PROGRAM MQTT
VAR
// Local Variables for Mqtt Client handling
	fbIotMqttClient : FB_IotMqttClient;
	bSetParameter 	: BOOL := TRUE;
	bConnect 		: BOOL := TRUE;	
	
// Publish message
	initMQTT : BOOL := FALSE;
	sTopicPubToPowerMgmt : STRING(255); //:= CONCAT('Robots/PowerMgmt/Robot_', INT_TO_STRING(.Var_HAWIno.Robot_Number)); 	// ToDo: Bisher ist die Nummer des HAWino fest kodiert
	sTopicPubToPowerMgmt_SOC : STRING(255);// := CONCAT('Robots/PowerMgmt/SoC_Robot_', INT_TO_STRING(.Var_HAWIno.Robot_Number)); 
	sPayloadPub : STRING(2000);	
	fbTimerPub 	: TON := (PT:=T#500MS);									// Intervall für das Senden des Akku-Status
	
//Received message
	bSubscribed    : BOOL;
	sTopicSubToPowerMgmt : STRING(255);// := CONCAT('PowerMgmt/Robots/Robot_', INT_TO_STRING(.Var_HAWIno.Robot_Number));	// ToDo: Bisher ist die Nummer des HAWino fest kodiert
	sTopicRcv      : STRING(255);
	sPayloadRcv    : STRING(255);
	sPayloadRcv_Status    : STRING(255);
	sPayloadRcv_Status_Test: STRING(255);
	fbMessageQueue : FB_IotMqttMessageQueue;
    fbMessage      : FB_IotMqttMessage;
	hrErrorOccurred : HRESULT; 			// Enthlt dern letzten augetretenen Fehler
	
//subscribe
	sTopicSubToGW1_Status : STRING(255);
	sTopicSubToGW1_Auftrag : STRING(255);
	sTopicSubCollision : STRING(255);
	sTopicPubCollision : ARRAY[1..4] OF STRING(255);
	sTopicSubReset : STRING(255);
	
// Variables for JSON
	fbJson			: FB_JsonSaxWriter;
	fbJsonDataType 	: FB_JsonReadWriteDataType;
	sJsonDoc       	: STRING(2000); 
	
// Local Variables for TwinCAT IoT Communication (TF6701) with direct link to EK1200 and TcCom
	//stMqtt_HAWino_In	AT%I*	: ST_PwrMgmt_HAWino_In;		// Attention! Don't link TIME Variables, otherwise we get an error!
	//stMqtt_HAWino_Out	AT%Q*	: ST_PwrMgmt_HAWino_Out;
	
	stMqtt_HAWino_In	 AT%I*: ST_PwrMgmt_HAWino_In;		// Attention! Don't link TIME Variables, otherwise we get an error!
	stMqtt_HAWino_Out	 AT%Q*: ST_PwrMgmt_HAWino_Out;
	
	SOC_Out : STRING(255);
	nBatteryTemperature	AT%I*	: INT;
	
	bComCheckAnswer	AT%Q*	: BOOL;
	
	stMqtt_HAWinoValues	: ST_PwrMgmt_HAWino;
	
	
// Timer to create a time stamp
	fbTimerTimestamp : TON := (PT:=T#71582M47S295MS);
	
// Local Vaiables to evaluate and act to input
	fbComCheckFlag	: RS;
	
	sTopicSubToFleetMgmt: STRING;
	Reset1: BOOL;
	//Input synccheck. robotdata has been read and can be used.
	txtReadInit AT%I* : BOOL := FALSE;
	
	//eigene Topics und Payload
	sTopicPubToGW1 : STRING(255);
	WerkstueckAusgelesen: BOOL;
	sPayloadPub1 : STRING(2000);
	Robotstatus : RobotStatusGW1;
	sTopicSubToGW1: STRING(255);
	nPayloadSize:INT;
	sPayloadPubCollision : STRING(100);
	n: INT;												
	
	FeedbackToGW1 AT%I*: STRING(50);				//Statusmeldungen an Gewerk 1
	RoboNmbToGoBack AT%I* : ARRAY[0..4] OF INT;		//Nummer, der Roboter, die zurück sollen
	resetVar, resetGoBack AT%I*: BOOL;				//Reset Variablen, um Ausgänge zurückzusetzen
	Auftrag AT%Q*: Auftrag;							//Auftrag von Gewerk 1 gesendet
	StatusFromGW1 AT%Q*: STRING(50);				//Statusrückmeldungen von Gewerk 1 gesendet
	goBack AT%Q* : BOOL;							//true, wenn Roboter Platz machen soll
	resetButton AT%Q* : BOOL;						//Reset von Gewerk 1 kommend
END_VAR

//Case machen! preop op

//Unsere Topics und erwartete Struktur:
//Auftrag: {"Art":"Fahrauftrag","AbholStation":1,"AbholTasche":2,"AblageStation":3,"AblageTasche":1}
//Status: {"Status":"WerkstueckAusgelesen"}
//Kollision: {"todo":"goBack"}

IF txtReadInit THEN
	IF NOT initMQTT THEN
		sTopicPubToPowerMgmt  := CONCAT('Robots/PowerMgmt/Robot_', INT_TO_STRING(.Var_HAWIno.Robot_Number)); 	
		sTopicPubToPowerMgmt_SOC  := CONCAT('Robots/PowerMgmt/SoC_Robot_', INT_TO_STRING(.Var_HAWIno.Robot_Number)); 
		sTopicSubToPowerMgmt  := CONCAT('PowerMgmt/Robots/Robot_', INT_TO_STRING(.Var_HAWIno.Robot_Number));
		sTopicSubToGW1  := CONCAT('VPJ/Robot_', INT_TO_STRING(.Var_HAWIno.Robot_Number));
		sTopicSubToGW1_Status  := CONCAT(sTopicSubToGW1, '/Status');
		sTopicSubToGW1_Auftrag  := CONCAT(sTopicSubToGW1, '/Auftrag');
		sTopicPubToGW1 := CONCAT('VPJ/Robot_', INT_TO_STRING(.Var_HAWIno.Robot_Number));
		sTopicSubCollision := CONCAT('VPJ/Robot_', INT_TO_STRING(.Var_HAWIno.Robot_Number));
		sTopicSubCollision := CONCAT(sTopicSubCollision, '/Collision');
		sTopicSubReset  := CONCAT('VPJ/Robot_', INT_TO_STRING(.Var_HAWIno.Robot_Number));
		sTopicSubReset  := CONCAT(sTopicSubToGW1, '/Reset');
		FOR n := 1 TO 4 BY 1 DO
			IF n <> .Var_HAWIno.Robot_Number THEN
				sTopicPubCollision[n] := CONCAT('VPJ/Robot_', INT_TO_STRING(n));
				sTopicPubCollision[n] := CONCAT(sTopicPubCollision[n], '/Collision');
			END_IF
		END_FOR
		initMQTT:= TRUE;
	END_IF
	
	stMqtt_HAWinoValues.Output.nRobotNumber := .Var_HAWIno.Robot_Number;			// Anpassen für jeden HAWino
	
	fbTimerTimestamp(In:= NOT fbTimerTimestamp.Q, ET=>stMqtt_HAWinoValues.Output.tTimestamp);
	
	stMqtt_HAWinoValues.Output.fSoC := stMqtt_HAWino_In.fSoC;
	
	stMqtt_HAWinoValues.Output.fActualBatteryCurrent := stMqtt_HAWino_In.fActualBatteryCurrent;
	stMqtt_HAWinoValues.Output.fActualBatteryVoltage := stMqtt_HAWino_In.fActualBatteryVoltage;

	
	// Skalierung der Temperaturwerte des Akkus
	stMqtt_HAWinoValues.Output.fBatteryTemperature := FKT_Scale(Rohwert := nBatteryTemperature, 
																	X1 := -500,
																	X2 := 1500, 
																	Y1 := -50,
																	Y2 := 150);
																	
	// Ausgabe der erwarteten Laufzeit des Roboters
	stMqtt_HAWinoValues.Output.nEstimatedRunningTime	:= LIMIT(0,stMqtt_HAWino_In.nEstimatedRunningTime,172800);		// Max. 48 Stunden sollen dargestellt werden
	stMqtt_HAWinoValues.Output.nEstimatedChargingTime	:= LIMIT(0,stMqtt_HAWino_In.nEstimatedChargingTime,172800);		// Max. 48 Stunden sollen dargestellt werden
	
	
	// Antworten auf den Kommunikationstest und des Ladetests
	stMqtt_HAWinoValues.Output.bCheckCurrentDetected := stMqtt_HAWino_In.bCheckCurrentDetected;
	stMqtt_HAWinoValues.Output.bComCheckAnswer := stMqtt_HAWino_In.bComCheckAnswer;
	
	//
	// Setting the parameters for establishing the connection to the Mqtt Broker and initializing the connection.
	//
	IF bSetParameter THEN
		fbIotMqttClient.sHostName := '192.168.0.11';	// IP-Adresse des Servers
		fbIotMqttClient.nHostPort := 1883;
		//fbIotMqttClient.sClientId := ClientId;
		fbIotMqttClient.sClientId := CONCAT('Robot_', INT_TO_STRING(.Var_HAWIno.Robot_Number));
		fbIotMqttClient.sTopicPrefix := '';
		//fbIotMqttClient.nKeepAlive:= 60; 
		fbIotMqttClient.sUserName:= 'VPJ';
		fbIotMqttClient.sUserPassword:= 'R462';
		//fbIotMqttClient.stWill:= ; 
		//fbIotMqttClient.stTLS:= ;
		fbIotMqttClient.ipMessageQueue := fbMessageQueue;
	
		bSetParameter := FALSE;
	END_IF
	
	
	//
	// This method -> MUST BE CALLED CYCLICALLY <- to ensure background communication with the MQTT broker.
	//
	fbIotMqttClient.Execute(bConnect);
	
	IF fbIotMqttClient.bError THEN
		// ToDo: add error logging here
		hrErrorOccurred := fbIotMqttClient.hrErrorCode;
	END_IF
	
		
	IF fbIotMqttClient.bConnected THEN		// Kontrolle, ob der Broker verbunden ist
		IF NOT bSubscribed THEN
			//
			// Abbonieren der Toopics, welche vom PowerMgmt kommen
			//
			bSubscribed := fbIotMqttClient.Subscribe(sTopic:=sTopicSubToPowerMgmt, eQoS:=TcIotMqttQos.AtMostOnceDelivery);
			IF fbIotMqttClient.bError THEN
				// ToDo: add my error logging here
				hrErrorOccurred := fbIotMqttClient.hrErrorCode;
			END_IF
			
			//
			// Abbonieren der Toopics, welche vom Gewerk 1 kommen
			//
			//Abbonieren von Topics: VPJ/Roboter
			bSubscribed := fbIotMqttClient.Subscribe(sTopic:=sTopicSubToGW1_Status, eQoS:=TcIotMqttQos.AtMostOnceDelivery);
			bSubscribed := fbIotMqttClient.Subscribe(sTopic:=sTopicSubToGW1_Auftrag, eQoS:=TcIotMqttQos.AtMostOnceDelivery);
			bSubscribed := fbIotMqttClient.Subscribe(sTopic:=sTopicSubCollision, eQoS:=TcIotMqttQos.AtMostOnceDelivery);
			bSubscribed := fbIotMqttClient.Subscribe(sTopic:=sTopicSubReset, eQoS:=TcIotMqttQos.AtMostOnceDelivery);
			
			
			//bSubscribed := fbIotMqttClient.Subscribe(sTopic:=sTopicSubToFleetMgmt, eQoS:=TcIotMqttQos.AtMostOnceDelivery);
			//IF fbIotMqttClient.bError THEN
				// ToDo: add my error logging here
			//	hrErrorOccurred := fbIotMqttClient.hrErrorCode;
			//END_IF
			
		END_IF
	END_IF	
	
	
	
	// Senden der MQTT- Nachrichten
	
	
	IF fbIotMqttClient.bConnected THEN			// Kontrolle, ob Broker verbunden ist
		fbTimerPub(IN:=TRUE);
		
		//
		// publish new paylod every 500 MS
		//
		IF fbTimerPub.Q THEN					// Abwarten des oben eingestellten Intervalls
			fbTimerPub(IN:=FALSE);
			
			//
			// Nachricht an PowerMgmt
			//
			fbJson.ResetDocument();
			fbJsonDataType.AddJsonValueFromSymbol(fbJson, 'ST_PwrMgmt_HAWino_In', SIZEOF(stMqtt_HAWinoValues.Output), ADR(stMqtt_HAWinoValues.Output));
			//sJsonDoc := fbJson.GetDocument();
			fbJson.CopyDocument(sJsonDoc, SIZEOF(sJsonDoc));
			
			sPayloadPub := sJsonDoc;	
			fbIotMqttClient.Publish(sTopic:= sTopicPubToPowerMgmt, 
										pPayload:= ADR(sPayloadPub), 
										nPayloadSize:= LEN2(ADR(sPayloadPub))+1, 										
										eQoS:= TcIotMqttQos.AtMostOnceDelivery, 
										bRetain:= FALSE, 
										bQueue:= FALSE);
									
									
			
			SOC_Out	:= CONCAT( '{"SoC" : ',LREAL_TO_STRING(stMqtt_HAWinoValues.Output.fSoC));
			SOC_Out	:= CONCAT( SOC_Out,'}');
			
			
			
			
			//SOC_Out := 	LREAL_TO_STRING(stMqtt_HAWinoValues.Output.fSoC);
			
						
			fbIotMqttClient.Publish(sTopic:= sTopicPubToPowerMgmt_SOC, 
										pPayload:=ADR(SOC_Out), 
										nPayloadSize:= INT_TO_UDINT(LEN(SOC_Out)),
										eQoS:= TcIotMqttQos.AtMostOnceDelivery, 
										bRetain:= FALSE, 
										bQueue:= FALSE);
										
										
			IF fbIotMqttClient.bError THEN
				// ToDo: add error logging here
				hrErrorOccurred := fbIotMqttClient.hrErrorCode;
			END_IF	
			
			//
			// Nachricht an GW1 - Produktionsauftrag
			//
			
			//Rückmeldung Roboterstatus
			sPayloadPub1 := CONCAT( '{"Status" : ', FeedbackToGW1);
			sPayloadPub1 := CONCAT( sPayloadPub1,'}');
			
			fbIotMqttClient.Publish(sTopic:= sTopicPubToGW1, 
											pPayload:=ADR(sPayloadPub1), 
											nPayloadSize:= INT_TO_UDINT(LEN(sPayloadPub1)),
											eQoS:= TcIotMqttQos.AtMostOnceDelivery, 
											bRetain:= FALSE, 
											bQueue:= FALSE);
											
			//An alle Roboter, die an Kollision beteiligt sind, goBack senden
			FOR n := 0 TO 4 BY 1 DO
				IF RoboNmbToGoBack[n] > 0 THEN
					sPayloadPubCollision := '{"todo":"goBack"}';
					
					fbIotMqttClient.Publish(sTopic:= sTopicPubCollision[RoboNmbToGoBack[n]], 
													pPayload:=ADR(sPayloadPubCollision), 
													nPayloadSize:= INT_TO_UDINT(LEN(sPayloadPubCollision)),
													eQoS:= TcIotMqttQos.AtMostOnceDelivery, 
													bRetain:= FALSE, 
													bQueue:= FALSE);
				END_IF
			END_FOR
		END_IF
	END_IF
	
	
	// Verarbeiten der Subscriptions
	
	
	IF fbMessageQueue.nQueuedMessages > 0 THEN			// Kontrolle, ob neue Daten vorliegen
		IF fbMessageQueue.Dequeue(fbMessage:=fbMessage) THEN
			fbMessage.GetTopic(pTopic:=ADR(sTopicRcv), nTopicSize:=SIZEOF(sTopicRcv) );
			

				
			//
			// Message from PowerMgmt
			//
			IF fbMessage.CompareTopic(sTopic:=sTopicSubToPowerMgmt) THEN		// Wenn die Daten vom PowerMgmt kommen, dann führe folgenede Aktion aus
				fbMessage.GetPayload(pPayload:=ADR(sPayloadRcv), nPayloadSize:=SIZEOF(sPayloadRcv), bSetNullTermination:=FALSE);
			// Json-String aufteilen und in Variablen schreiben
				fbJsonDataType.SetSymbolFromJson(sPayloadRcv,'ST_PwrMgmt_HAWino_Out',SIZEOF(stMqtt_HAWinoValues.Input),ADR(stMqtt_HAWinoValues.Input));
			END_IF
		
			//
			// Hier werden weitere Topics verarbeitet
			// 
			//Status von Gewerk 1 kommend
			IF fbMessage.CompareTopic(sTopic:=sTopicSubToGW1_Status) THEN
				
				fbMessage.GetPayload(pPayload:=ADR(sPayloadRcv_Status), nPayloadSize:=SIZEOF(sPayloadRcv_Status), bSetNullTermination:=true);
				// Json-String aufteilen und in Variablen schreiben
				fbJsonDataType.SetSymbolFromJson(sPayloadRcv_Status,'RobotStatusGW1',SIZEOF(RobotStatus),ADR(RobotStatus));
				StatusFromGW1 := Robotstatus.Status;
				Robotstatus.Status := '';
				sPayloadRcv_Status := '';
			END_IF
			
			//Auftrag von Gewerk 1 kommend
			IF fbMessage.CompareTopic(sTopic:=sTopicSubToGW1_Auftrag) THEN
				fbMessage.GetPayload(pPayload:=ADR(sPayloadRcv), nPayloadSize:=SIZEOF(sPayloadRcv), bSetNullTermination:=TRUE);
			
			// Json-String aufteilen und in Variablen schreiben
				fbJsonDataType.SetSymbolFromJson(sPayloadRcv,'Auftrag',SIZEOF(Auftrag),ADR(Auftrag));
			END_IF
			
			//Nachricht von anderem HAWino, dass dieser zurückfahren soll
			IF fbMessage.CompareTopic(sTopic:=sTopicSubCollision) THEN
				goBack := TRUE;
			END_IF
			
			//Nachricht von Gewerk 1, dass HAWino reset machen soll (nach Fehler)
			IF fbMessage.CompareTopic(sTopic:=sTopicSubReset) THEN
				resetButton := TRUE;
			END_IF
			
		END_IF
	END_IF	
	
	//Rücksetzen der durch Gewerk 1 beschriebenen Variablen
	IF resetVar THEN
		StatusFromGW1 := '';
		Robotstatus.Status := '';
		sPayloadRcv_Status := '';
		Auftrag.AbholStation := 0;
		Auftrag.AbholTasche := 0;
		Auftrag.AblageStation := 0;
		Auftrag.AblageTasche := 0;
		Auftrag.Art := '';
		resetButton := FALSE;
	END_IF
	
	IF resetGoBack THEN
		goBack := FALSE;
	END_IF
	
	
	// Evaulierung der empfangenen Daten
	
	//
	// ToDo: Plausibilitätsprüfung von stMqtt_HAWinoValues.Input und evt. TypConversion
	// Attention! The assignment of input to output is correct. Don `t change!
	//	
	
	stMqtt_HAWino_Out.bChargingActive := stMqtt_HAWinoValues.Input.bChargingActive;
	stMqtt_HAWino_Out.bExternalRecalibrationTrigger := stMqtt_HAWinoValues.Input.bExternalRecalibrationTrigger;
	stMqtt_HAWino_Out.fExternalRecalibrationValue := stMqtt_HAWinoValues.Input.fExternalRecalibrationValue;
	
	
	// Hier Communication Check einbauen
	
	//fbComCheckFlag(Set:= stMqtt_HAWinoValues.Input.bComCheckRequest, 
	//					Reset1:= NOT stMqtt_HAWinoValues.Input.bComCheckRequest,
	//					Q1 => bComCheckAnswer);
	bComCheckAnswer	:= TRUE;
					
END_IF

END_PROGRAM

(* stored: Version 1.1.0.1, ProductVersion 3.1.4024.11
   POU MQTT: Id {3b364ef0-24c5-4b55-9f63-1e0f62f8b4d0}, SpecialFunc None *)
